FUNCTION_BLOCK Pallet_HMI
  (* Standard: 61499-2 *)
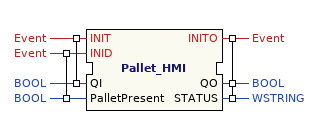
  EVENT_INPUT
    INIT WITH QI;
    INID WITH PalletPresent;
  END_EVENT
  EVENT_OUTPUT
    INITO WITH QO, STATUS;
  END_EVENT
  VAR_INPUT
    QI : BOOL;
    PalletPresent : BOOL;
  END_VAR
  VAR_OUTPUT
    QO : BOOL;
    STATUS : WSTRING;
  END_VAR
END_FUNCTION_BLOCK
